// TIA Portal V21 export
VAR_GLOBAL   // PLC tag table "UnitàDiMisura_Tipi"
END_VAR
VAR_GLOBAL CONSTANT   // user constants
   Um_TipoLunghezza_Metri : Int := 1;
   Um_TipoLunghezza_Piedi : Int := 2;
   Um_TipoLunghezza_Pollici : Int := 3;
   Um_TipoPercentuale_Perc : Int := 1;
   "Um_TipoTemperatura_°C" : Int := 1;
   "Um_TipoTemperatura_°F" : Int := 2;
   Um_TipoTemperatura_Kelvin : Int := 3;
   Um_TipoPortata_Metricubi : Int := 1;
   Um_TipoPortata_Litri : Int := 2;
   Um_TipoPressione_Bar : Int := 1;
   Um_TipoPressione_PSI : Int := 2;
   Um_TipoPressione_Atmosfera : Int := 3;
   "Um_TipoConcentrazione_mg/l" : Int := 1;
END_VAR
